TYPE sPositions :
STRUCT
	reX : REAL;       // X-Position
	reY : REAL;       // Y-Position
	reWinkel : REAL; // Ausrichtung
END_STRUCT
END_TYPE

(* stored: Version 1.1.0.1, ProductVersion 3.1.4026.13
   DUT sPositions: Id {bfef0853-728b-4fd4-b0c4-5120a61fcf44} *)
